// Mitsubishi GX Works2 project: GAO-71UR-20100027-0427R   PLC: Q00U

PROGRAM MAIN
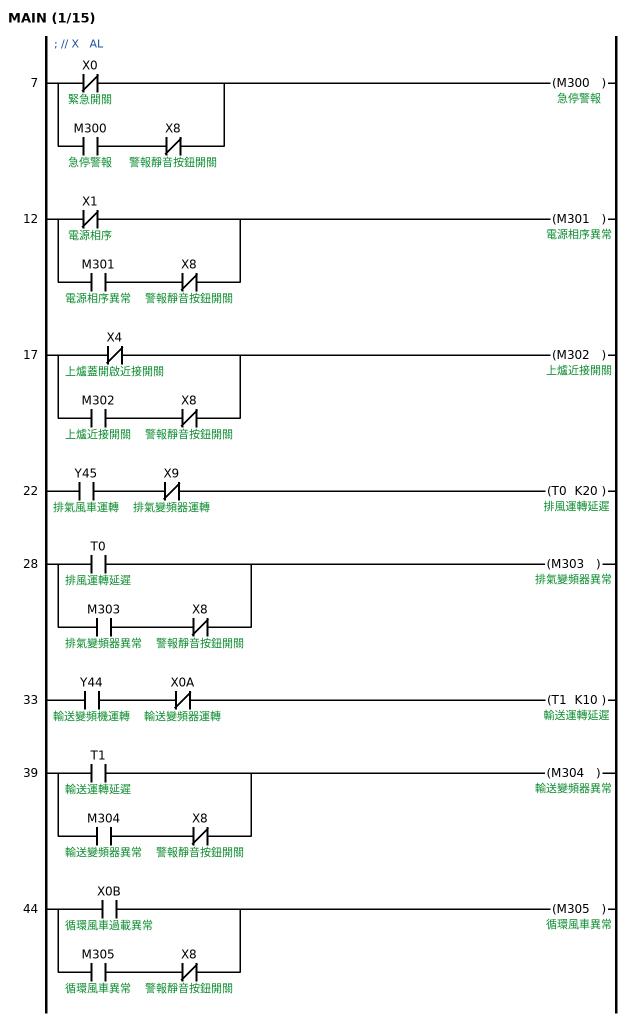
; // X   AL
7     LDI     X0  ; 緊急開關
      LD      M300  ; 急停警報
      ANI     X8  ; 警報靜音按鈕開關
      ORB
      OUT     M300  ; 急停警報
12    LDI     X1  ; 電源相序
      LD      M301  ; 電源相序異常
      ANI     X8  ; 警報靜音按鈕開關
      ORB
      OUT     M301  ; 電源相序異常
17    LDI     X4  ; 上爐蓋開啟近接開關
      LD      M302  ; 上爐近接開關
      ANI     X8  ; 警報靜音按鈕開關
      ORB
      OUT     M302  ; 上爐近接開關
22    LD      Y45  ; 排氣風車運轉
      ANI     X9  ; 排氣變頻器運轉
      OUT     T0 K20  ; 排風運轉延遲
28    LD      T0  ; 排風運轉延遲
      LD      M303  ; 排氣變頻器異常
      ANI     X8  ; 警報靜音按鈕開關
      ORB
      OUT     M303  ; 排氣變頻器異常
33    LD      Y44  ; 輸送變頻機運轉
      ANI     X0A  ; 輸送變頻器運轉
      OUT     T1 K10  ; 輸送運轉延遲
39    LD      T1  ; 輸送運轉延遲
      LD      M304  ; 輸送變頻器異常
      ANI     X8  ; 警報靜音按鈕開關
      ORB
      OUT     M304  ; 輸送變頻器異常
44    LD      X0B  ; 循環風車過載異常
      LD      M305  ; 循環風車異常
      ANI     X8  ; 警報靜音按鈕開關
      ORB
      OUT     M305  ; 循環風車異常
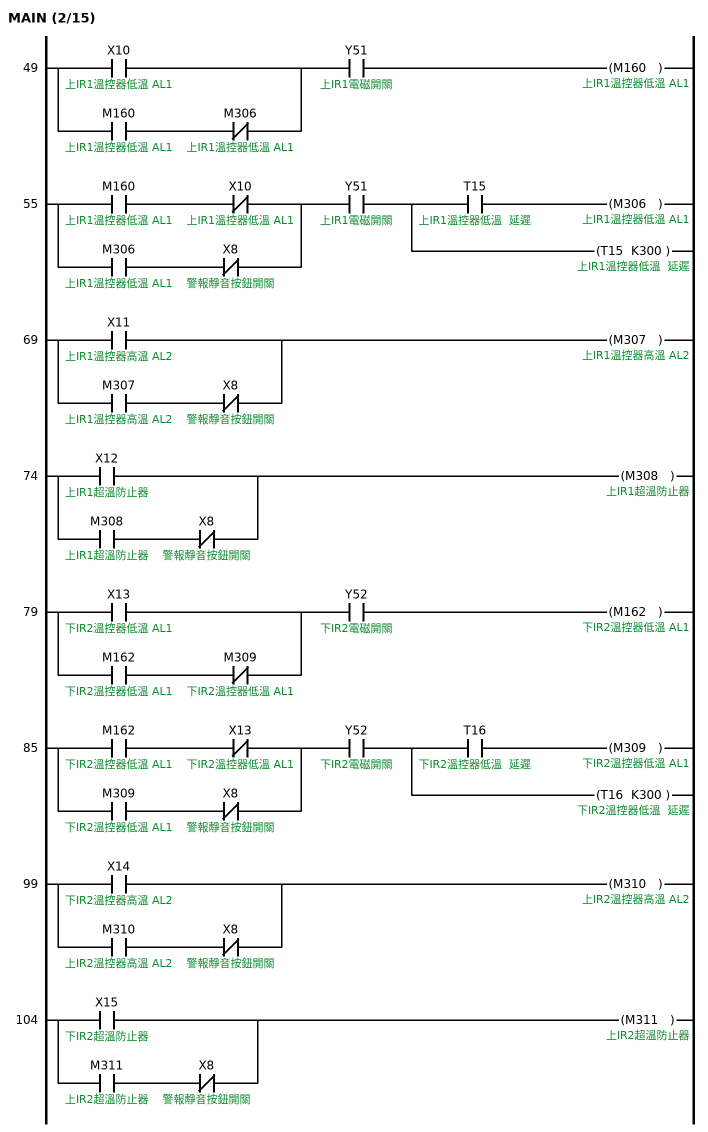
49    LD      X10  ; 上IR1溫控器低溫 AL1
      LD      M160  ; 上IR1溫控器低溫 AL1
      ANI     M306  ; 上IR1溫控器低溫 AL1
      ORB
      AND     Y51  ; 上IR1電磁開關
      OUT     M160  ; 上IR1溫控器低溫 AL1
55    LD      M160  ; 上IR1溫控器低溫 AL1
      ANI     X10  ; 上IR1溫控器低溫 AL1
      LD      M306  ; 上IR1溫控器低溫 AL1
      ANI     X8  ; 警報靜音按鈕開關
      ORB
      AND     Y51  ; 上IR1電磁開關
      MPS
      AND     T15  ; 上IR1溫控器低溫  延遲
      OUT     M306  ; 上IR1溫控器低溫 AL1
      MPP
      OUT     T15 K300  ; 上IR1溫控器低溫  延遲
69    LD      X11  ; 上IR1溫控器高溫 AL2
      LD      M307  ; 上IR1溫控器高溫 AL2
      ANI     X8  ; 警報靜音按鈕開關
      ORB
      OUT     M307  ; 上IR1溫控器高溫 AL2
74    LD      X12  ; 上IR1超溫防止器
      LD      M308  ; 上IR1超溫防止器
      ANI     X8  ; 警報靜音按鈕開關
      ORB
      OUT     M308  ; 上IR1超溫防止器
79    LD      X13  ; 下IR2溫控器低溫 AL1
      LD      M162  ; 下IR2溫控器低溫 AL1
      ANI     M309  ; 下IR2溫控器低溫 AL1
      ORB
      AND     Y52  ; 下IR2電磁開關
      OUT     M162  ; 下IR2溫控器低溫 AL1
85    LD      M162  ; 下IR2溫控器低溫 AL1
      ANI     X13  ; 下IR2溫控器低溫 AL1
      LD      M309  ; 下IR2溫控器低溫 AL1
      ANI     X8  ; 警報靜音按鈕開關
      ORB
      AND     Y52  ; 下IR2電磁開關
      MPS
      AND     T16  ; 下IR2溫控器低溫  延遲
      OUT     M309  ; 下IR2溫控器低溫 AL1
      MPP
      OUT     T16 K300  ; 下IR2溫控器低溫  延遲
99    LD      X14  ; 下IR2溫控器高溫 AL2
      LD      M310  ; 上IR2溫控器高溫 AL2
      ANI     X8  ; 警報靜音按鈕開關
      ORB
      OUT     M310  ; 上IR2溫控器高溫 AL2
104   LD      X15  ; 下IR2超溫防止器
      LD      M311  ; 上IR2超溫防止器
      ANI     X8  ; 警報靜音按鈕開關
      ORB
      OUT     M311  ; 上IR2超溫防止器
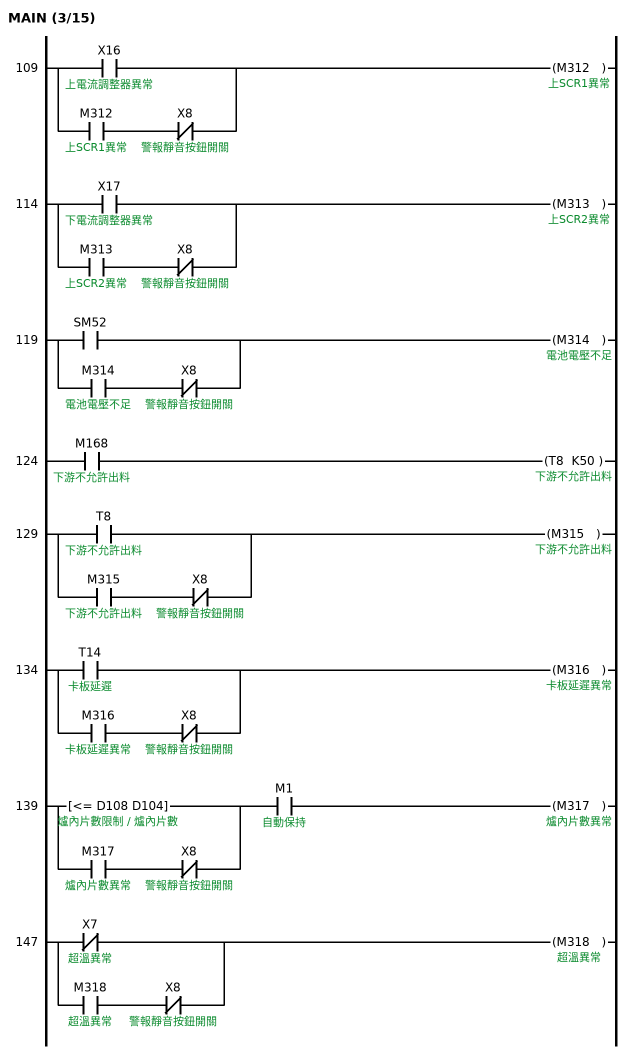
109   LD      X16  ; 上電流調整器異常
      LD      M312  ; 上SCR1異常
      ANI     X8  ; 警報靜音按鈕開關
      ORB
      OUT     M312  ; 上SCR1異常
114   LD      X17  ; 下電流調整器異常
      LD      M313  ; 上SCR2異常
      ANI     X8  ; 警報靜音按鈕開關
      ORB
      OUT     M313  ; 上SCR2異常
119   LD      SM52
      LD      M314  ; 電池電壓不足
      ANI     X8  ; 警報靜音按鈕開關
      ORB
      OUT     M314  ; 電池電壓不足
124   LD      M168  ; 下游不允許出料
      OUT     T8 K50  ; 下游不允許出料
129   LD      T8  ; 下游不允許出料
      LD      M315  ; 下游不允許出料
      ANI     X8  ; 警報靜音按鈕開關
      ORB
      OUT     M315  ; 下游不允許出料
134   LD      T14  ; 卡板延遲
      LD      M316  ; 卡板延遲異常
      ANI     X8  ; 警報靜音按鈕開關
      ORB
      OUT     M316  ; 卡板延遲異常
139   LD<=    D108 D104  ; 爐內片數限制 / 爐內片數
      LD      M317  ; 爐內片數異常
      ANI     X8  ; 警報靜音按鈕開關
      ORB
      AND     M1  ; 自動保持
      OUT     M317  ; 爐內片數異常
147   LDI     X7  ; 超溫異常
      LD      M318  ; 超溫異常
      ANI     X8  ; 警報靜音按鈕開關
      ORB
      OUT     M318  ; 超溫異常
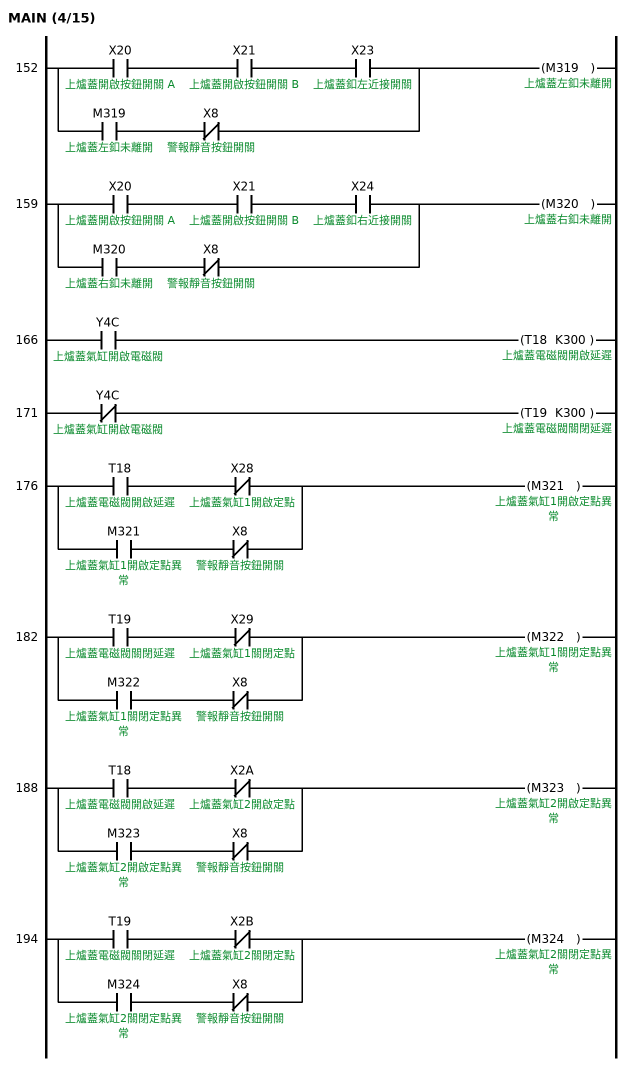
152   LD      X20  ; 上爐蓋開啟按鈕開關 A
      AND     X21  ; 上爐蓋開啟按鈕開關 B
      AND     X23  ; 上爐蓋釦左近接開關
      LD      M319  ; 上爐蓋左釦未離開
      ANI     X8  ; 警報靜音按鈕開關
      ORB
      OUT     M319  ; 上爐蓋左釦未離開
159   LD      X20  ; 上爐蓋開啟按鈕開關 A
      AND     X21  ; 上爐蓋開啟按鈕開關 B
      AND     X24  ; 上爐蓋釦右近接開關
      LD      M320  ; 上爐蓋右釦未離開
      ANI     X8  ; 警報靜音按鈕開關
      ORB
      OUT     M320  ; 上爐蓋右釦未離開
166   LD      Y4C  ; 上爐蓋氣缸開啟電磁閥
      OUT     T18 K300  ; 上爐蓋電磁閥開啟延遲
171   LDI     Y4C  ; 上爐蓋氣缸開啟電磁閥
      OUT     T19 K300  ; 上爐蓋電磁閥關閉延遲
176   LD      T18  ; 上爐蓋電磁閥開啟延遲
      ANI     X28  ; 上爐蓋氣缸1開啟定點
      LD      M321  ; 上爐蓋氣缸1開啟定點異常
      ANI     X8  ; 警報靜音按鈕開關
      ORB
      OUT     M321  ; 上爐蓋氣缸1開啟定點異常
182   LD      T19  ; 上爐蓋電磁閥關閉延遲
      ANI     X29  ; 上爐蓋氣缸1關閉定點
      LD      M322  ; 上爐蓋氣缸1關閉定點異常
      ANI     X8  ; 警報靜音按鈕開關
      ORB
      OUT     M322  ; 上爐蓋氣缸1關閉定點異常
188   LD      T18  ; 上爐蓋電磁閥開啟延遲
      ANI     X2A  ; 上爐蓋氣缸2開啟定點
      LD      M323  ; 上爐蓋氣缸2開啟定點異常
      ANI     X8  ; 警報靜音按鈕開關
      ORB
      OUT     M323  ; 上爐蓋氣缸2開啟定點異常
194   LD      T19  ; 上爐蓋電磁閥關閉延遲
      ANI     X2B  ; 上爐蓋氣缸2關閉定點
      LD      M324  ; 上爐蓋氣缸2關閉定點異常
      ANI     X8  ; 警報靜音按鈕開關
      ORB
      OUT     M324  ; 上爐蓋氣缸2關閉定點異常
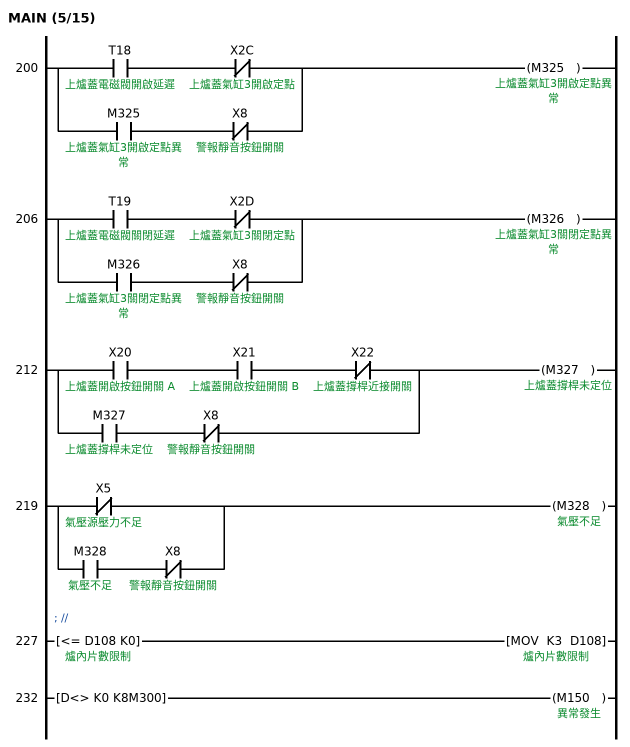
200   LD      T18  ; 上爐蓋電磁閥開啟延遲
      ANI     X2C  ; 上爐蓋氣缸3開啟定點
      LD      M325  ; 上爐蓋氣缸3開啟定點異常
      ANI     X8  ; 警報靜音按鈕開關
      ORB
      OUT     M325  ; 上爐蓋氣缸3開啟定點異常
206   LD      T19  ; 上爐蓋電磁閥關閉延遲
      ANI     X2D  ; 上爐蓋氣缸3關閉定點
      LD      M326  ; 上爐蓋氣缸3關閉定點異常
      ANI     X8  ; 警報靜音按鈕開關
      ORB
      OUT     M326  ; 上爐蓋氣缸3關閉定點異常
212   LD      X20  ; 上爐蓋開啟按鈕開關 A
      AND     X21  ; 上爐蓋開啟按鈕開關 B
      ANI     X22  ; 上爐蓋撐桿近接開關
      LD      M327  ; 上爐蓋撐桿未定位
      ANI     X8  ; 警報靜音按鈕開關
      ORB
      OUT     M327  ; 上爐蓋撐桿未定位
219   LDI     X5  ; 氣壓源壓力不足
      LD      M328  ; 氣壓不足
      ANI     X8  ; 警報靜音按鈕開關
      ORB
      OUT     M328  ; 氣壓不足
; //
227   LD<=    D108 K0  ; 爐內片數限制
      MOV     K3 D108
232   LDD<>   K0 K8M300  ; 急停警報
      OUT     M150  ; 異常發生
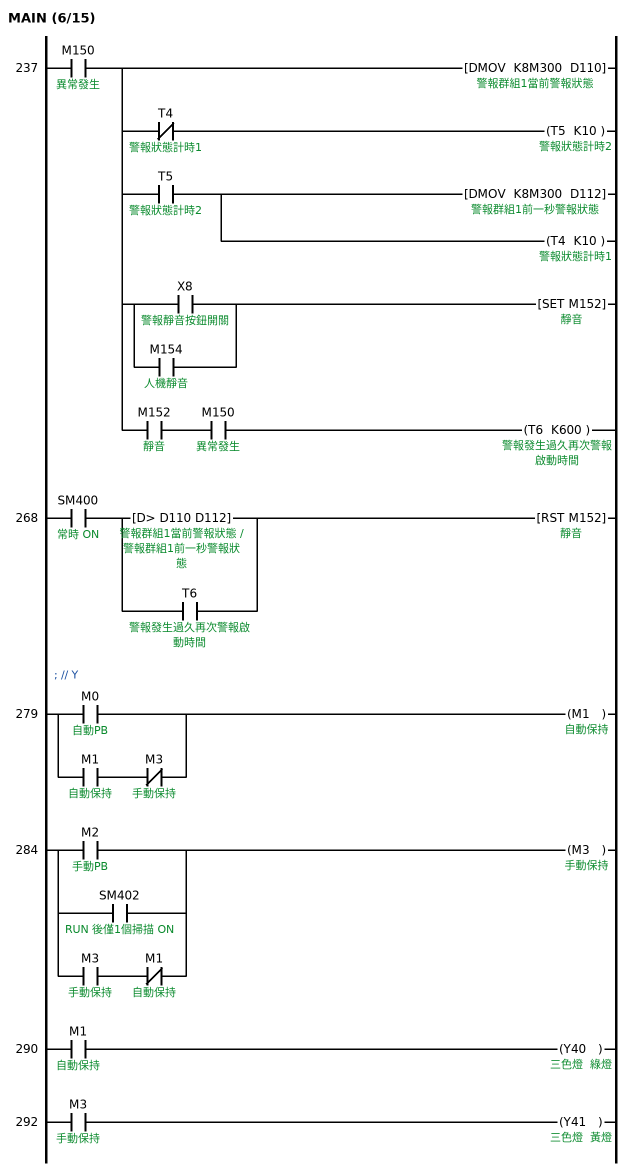
237   LD      M150  ; 異常發生
      DMOV    K8M300 D110  ; 警報群組1當前警報狀態
      MPS
      ANI     T4  ; 警報狀態計時1
      OUT     T5 K10  ; 警報狀態計時2
      MRD
      AND     T5  ; 警報狀態計時2
      DMOV    K8M300 D112  ; 警報群組1前一秒警報狀態
      OUT     T4 K10  ; 警報狀態計時1
      MRD
      LD      X8  ; 警報靜音按鈕開關
      OR      M154  ; 人機靜音
      ANB
      SET     M152  ; 靜音
      MPP
      AND     M152  ; 靜音
      AND     M150  ; 異常發生
      OUT     T6 K600  ; 警報發生過久再次警報啟動時間
268   LD      SM400  ; 常時 ON
      LDD>    D110 D112  ; 警報群組1當前警報狀態 / 警報群組1前一秒警報狀態
      OR      T6  ; 警報發生過久再次警報啟動時間
      ANB
      RST     M152  ; 靜音
; // Y
279   LD      M0  ; 自動PB
      LD      M1  ; 自動保持
      ANI     M3  ; 手動保持
      ORB
      OUT     M1  ; 自動保持
284   LD      M2  ; 手動PB
      OR      SM402  ; RUN 後僅1個掃描 ON
      LD      M3  ; 手動保持
      ANI     M1  ; 自動保持
      ORB
      OUT     M3  ; 手動保持
290   LD      M1  ; 自動保持
      OUT     Y40  ; 三色燈  綠燈
292   LD      M3  ; 手動保持
      OUT     Y41  ; 三色燈  黃燈
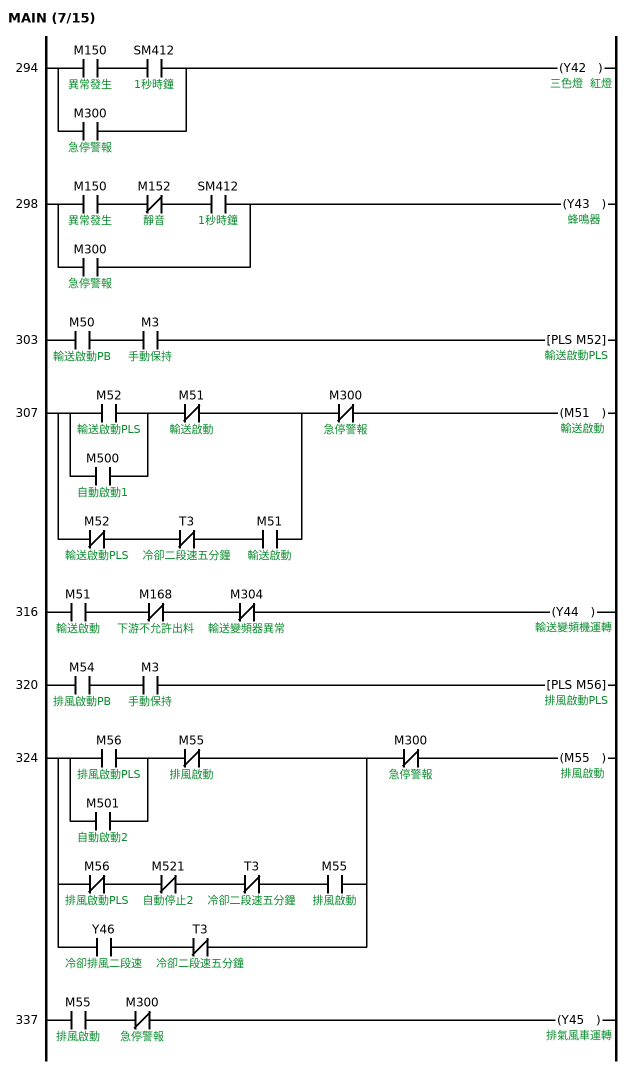
294   LD      M150  ; 異常發生
      AND     SM412  ; 1秒時鐘
      OR      M300  ; 急停警報
      OUT     Y42  ; 三色燈  紅燈
298   LD      M150  ; 異常發生
      ANI     M152  ; 靜音
      AND     SM412  ; 1秒時鐘
      OR      M300  ; 急停警報
      OUT     Y43  ; 蜂鳴器
303   LD      M50  ; 輸送啟動PB
      AND     M3  ; 手動保持
      PLS     M52  ; 輸送啟動PLS
307   LD      M52  ; 輸送啟動PLS
      OR      M500  ; 自動啟動1
      ANI     M51  ; 輸送啟動
      LDI     M52  ; 輸送啟動PLS
      ANI     T3  ; 冷卻二段速五分鐘
      AND     M51  ; 輸送啟動
      ORB
      ANI     M300  ; 急停警報
      OUT     M51  ; 輸送啟動
316   LD      M51  ; 輸送啟動
      ANI     M168  ; 下游不允許出料
      ANI     M304  ; 輸送變頻器異常
      OUT     Y44  ; 輸送變頻機運轉
320   LD      M54  ; 排風啟動PB
      AND     M3  ; 手動保持
      PLS     M56  ; 排風啟動PLS
324   LD      M56  ; 排風啟動PLS
      OR      M501  ; 自動啟動2
      ANI     M55  ; 排風啟動
      LDI     M56  ; 排風啟動PLS
      ANI     M521  ; 自動停止2
      ANI     T3  ; 冷卻二段速五分鐘
      AND     M55  ; 排風啟動
      ORB
      LD      Y46  ; 冷卻排風二段速
      ANI     T3  ; 冷卻二段速五分鐘
      ORB
      ANI     M300  ; 急停警報
      OUT     M55  ; 排風啟動
337   LD      M55  ; 排風啟動
      ANI     M300  ; 急停警報
      OUT     Y45  ; 排氣風車運轉
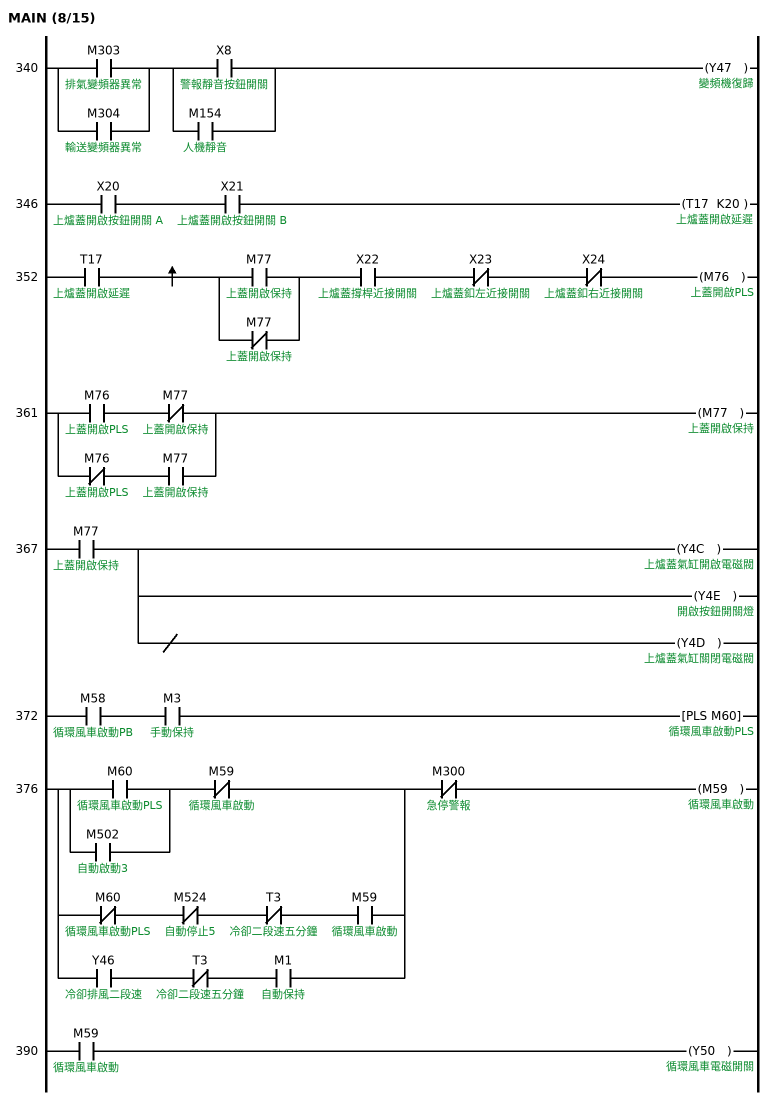
340   LD      M303  ; 排氣變頻器異常
      OR      M304  ; 輸送變頻器異常
      LD      X8  ; 警報靜音按鈕開關
      OR      M154  ; 人機靜音
      ANB
      OUT     Y47  ; 變頻機復歸
346   LD      X20  ; 上爐蓋開啟按鈕開關 A
      AND     X21  ; 上爐蓋開啟按鈕開關 B
      OUT     T17 K20  ; 上爐蓋開啟延遲
352   LD      T17  ; 上爐蓋開啟延遲
      MEP
      LD      M77  ; 上蓋開啟保持
      ORI     M77  ; 上蓋開啟保持
      ANB
      AND     X22  ; 上爐蓋撐桿近接開關
      ANI     X23  ; 上爐蓋釦左近接開關
      ANI     X24  ; 上爐蓋釦右近接開關
      OUT     M76  ; 上蓋開啟PLS
361   LD      M76  ; 上蓋開啟PLS
      ANI     M77  ; 上蓋開啟保持
      LDI     M76  ; 上蓋開啟PLS
      AND     M77  ; 上蓋開啟保持
      ORB
      OUT     M77  ; 上蓋開啟保持
367   LD      M77  ; 上蓋開啟保持
      OUT     Y4C  ; 上爐蓋氣缸開啟電磁閥
      OUT     Y4E  ; 開啟按鈕開關燈
      INV
      OUT     Y4D  ; 上爐蓋氣缸關閉電磁閥
372   LD      M58  ; 循環風車啟動PB
      AND     M3  ; 手動保持
      PLS     M60  ; 循環風車啟動PLS
376   LD      M60  ; 循環風車啟動PLS
      OR      M502  ; 自動啟動3
      ANI     M59  ; 循環風車啟動
      LDI     M60  ; 循環風車啟動PLS
      ANI     M524  ; 自動停止5
      ANI     T3  ; 冷卻二段速五分鐘
      AND     M59  ; 循環風車啟動
      ORB
      LD      Y46  ; 冷卻排風二段速
      ANI     T3  ; 冷卻二段速五分鐘
      AND     M1  ; 自動保持
      ORB
      ANI     M300  ; 急停警報
      OUT     M59  ; 循環風車啟動
390   LD      M59  ; 循環風車啟動
      OUT     Y50  ; 循環風車電磁開關
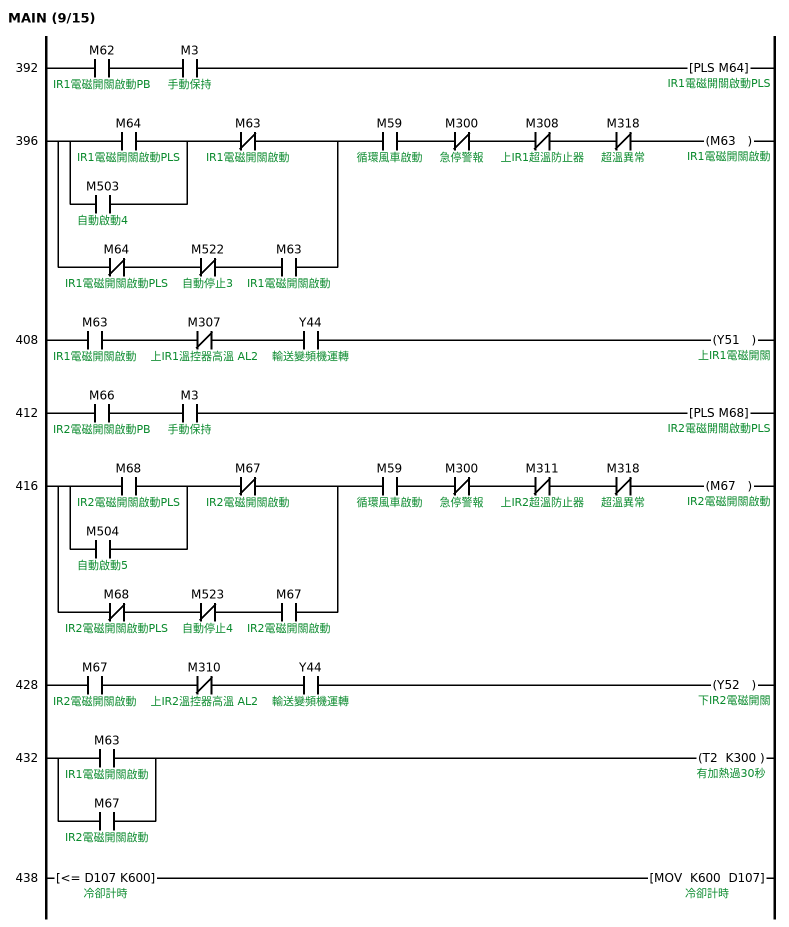
392   LD      M62  ; IR1電磁開關啟動PB
      AND     M3  ; 手動保持
      PLS     M64  ; IR1電磁開關啟動PLS
396   LD      M64  ; IR1電磁開關啟動PLS
      OR      M503  ; 自動啟動4
      ANI     M63  ; IR1電磁開關啟動
      LDI     M64  ; IR1電磁開關啟動PLS
      ANI     M522  ; 自動停止3
      AND     M63  ; IR1電磁開關啟動
      ORB
      AND     M59  ; 循環風車啟動
      ANI     M300  ; 急停警報
      ANI     M308  ; 上IR1超溫防止器
      ANI     M318  ; 超溫異常
      OUT     M63  ; IR1電磁開關啟動
408   LD      M63  ; IR1電磁開關啟動
      ANI     M307  ; 上IR1溫控器高溫 AL2
      AND     Y44  ; 輸送變頻機運轉
      OUT     Y51  ; 上IR1電磁開關
412   LD      M66  ; IR2電磁開關啟動PB
      AND     M3  ; 手動保持
      PLS     M68  ; IR2電磁開關啟動PLS
416   LD      M68  ; IR2電磁開關啟動PLS
      OR      M504  ; 自動啟動5
      ANI     M67  ; IR2電磁開關啟動
      LDI     M68  ; IR2電磁開關啟動PLS
      ANI     M523  ; 自動停止4
      AND     M67  ; IR2電磁開關啟動
      ORB
      AND     M59  ; 循環風車啟動
      ANI     M300  ; 急停警報
      ANI     M311  ; 上IR2超溫防止器
      ANI     M318  ; 超溫異常
      OUT     M67  ; IR2電磁開關啟動
428   LD      M67  ; IR2電磁開關啟動
      ANI     M310  ; 上IR2溫控器高溫 AL2
      AND     Y44  ; 輸送變頻機運轉
      OUT     Y52  ; 下IR2電磁開關
432   LD      M63  ; IR1電磁開關啟動
      OR      M67  ; IR2電磁開關啟動
      OUT     T2 K300  ; 有加熱過30秒
438   LD<=    D107 K600  ; 冷卻計時
      MOV     K600 D107
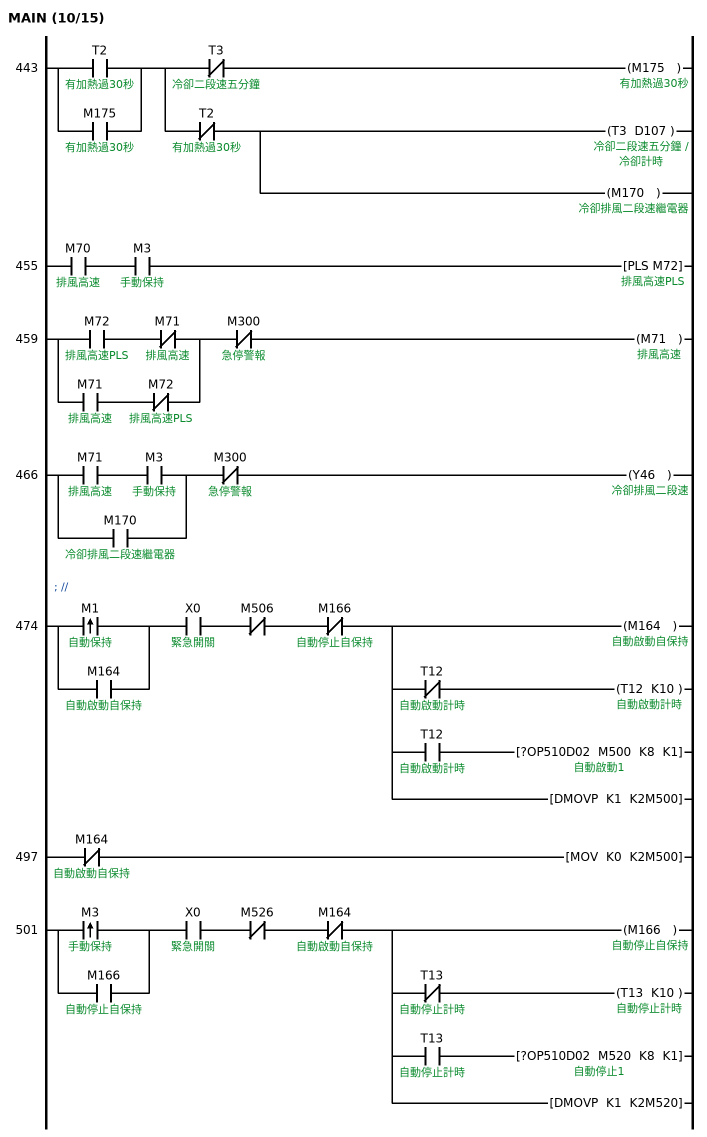
443   LD      T2  ; 有加熱過30秒
      OR      M175  ; 有加熱過30秒
      MPS
      ANI     T3  ; 冷卻二段速五分鐘
      OUT     M175  ; 有加熱過30秒
      MPP
      ANI     T2  ; 有加熱過30秒
      OUT     T3 D107  ; 冷卻二段速五分鐘 / 冷卻計時
      OUT     M170  ; 冷卻排風二段速繼電器
455   LD      M70  ; 排風高速
      AND     M3  ; 手動保持
      PLS     M72  ; 排風高速PLS
459   LD      M72  ; 排風高速PLS
      ANI     M71  ; 排風高速
      LD      M71  ; 排風高速
      ANI     M72  ; 排風高速PLS
      ORB
      ANI     M300  ; 急停警報
      OUT     M71  ; 排風高速
466   LD      M71  ; 排風高速
      AND     M3  ; 手動保持
      OR      M170  ; 冷卻排風二段速繼電器
      ANI     M300  ; 急停警報
      OUT     Y46  ; 冷卻排風二段速
; //
474   LDP     M1  ; 自動保持
      OR      M164  ; 自動啟動自保持
      AND     X0  ; 緊急開關
      ANI     M506
      ANI     M166  ; 自動停止自保持
      OUT     M164  ; 自動啟動自保持
      MPS
      ANI     T12  ; 自動啟動計時
      OUT     T12 K10  ; 自動啟動計時
      MRD
      AND     T12  ; 自動啟動計時
      ?OP510D02 M500 K8 K1
      MPP
      DMOVP   K1 K2M500
497   LDI     M164  ; 自動啟動自保持
      MOV     K0 K2M500
501   LDP     M3  ; 手動保持
      OR      M166  ; 自動停止自保持
      AND     X0  ; 緊急開關
      ANI     M526
      ANI     M164  ; 自動啟動自保持
      OUT     M166  ; 自動停止自保持
      MPS
      ANI     T13  ; 自動停止計時
      OUT     T13 K10  ; 自動停止計時
      MRD
      AND     T13  ; 自動停止計時
      ?OP510D02 M520 K8 K1  ; 自動停止1
      MPP
      DMOVP   K1 K2M520
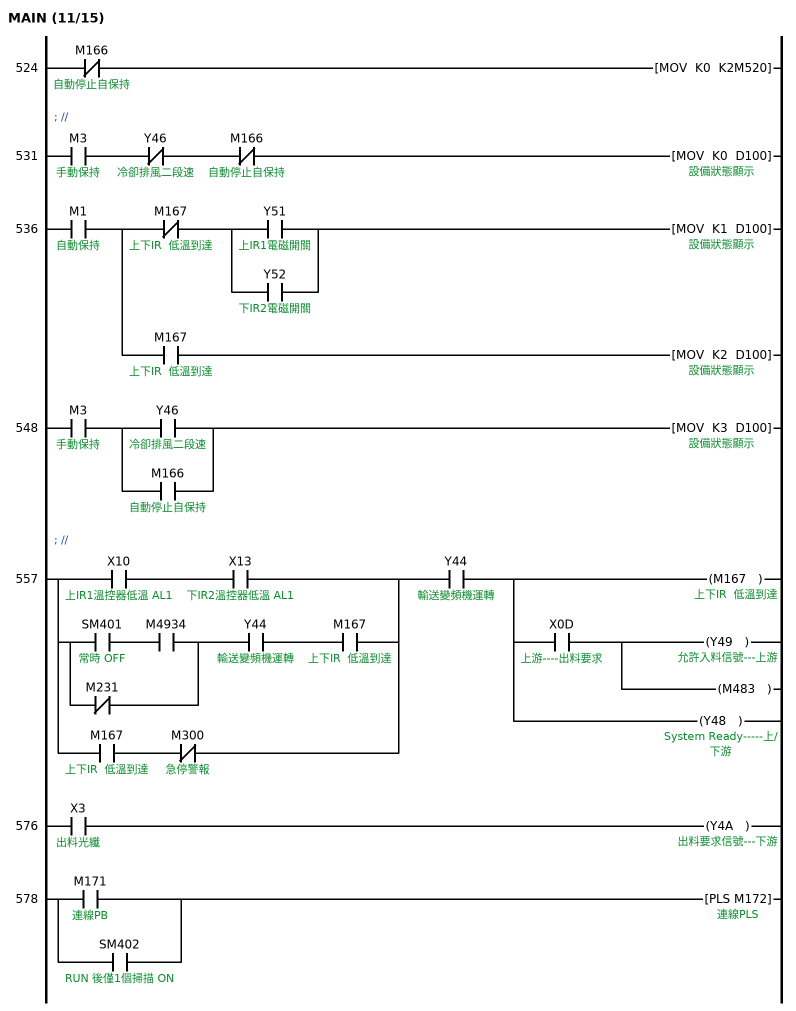
524   LDI     M166  ; 自動停止自保持
      MOV     K0 K2M520
; //
531   LD      M3  ; 手動保持
      ANI     Y46  ; 冷卻排風二段速
      ANI     M166  ; 自動停止自保持
      MOV     K0 D100  ; 設備狀態顯示
536   LD      M1  ; 自動保持
      MPS
      ANI     M167  ; 上下IR  低溫到達
      LD      Y51  ; 上IR1電磁開關
      OR      Y52  ; 下IR2電磁開關
      ANB
      MOV     K1 D100
      MPP
      AND     M167  ; 上下IR  低溫到達
      MOV     K2 D100
548   LD      M3  ; 手動保持
      LD      Y46  ; 冷卻排風二段速
      OR      M166  ; 自動停止自保持
      ANB
      MOV     K3 D100
; //
557   LD      X10  ; 上IR1溫控器低溫 AL1
      AND     X13  ; 下IR2溫控器低溫 AL1
      LD      SM401  ; 常時 OFF
      AND     M4934
      ORI     M231
      AND     Y44  ; 輸送變頻機運轉
      AND     M167  ; 上下IR  低溫到達
      ORB
      LD      M167  ; 上下IR  低溫到達
      ANI     M300  ; 急停警報
      ORB
      AND     Y44  ; 輸送變頻機運轉
      OUT     M167  ; 上下IR  低溫到達
      MPS
      AND     X0D  ; 上游----出料要求
      OUT     Y49  ; 允許入料信號---上游
      OUT     M483
      MPP
      OUT     Y48  ; System Ready-----上/下游
576   LD      X3  ; 出料光纖
      OUT     Y4A  ; 出料要求信號---下游
578   LD      M171  ; 連線PB
      OR      SM402  ; RUN 後僅1個掃描 ON
      PLS     M172  ; 連線PLS
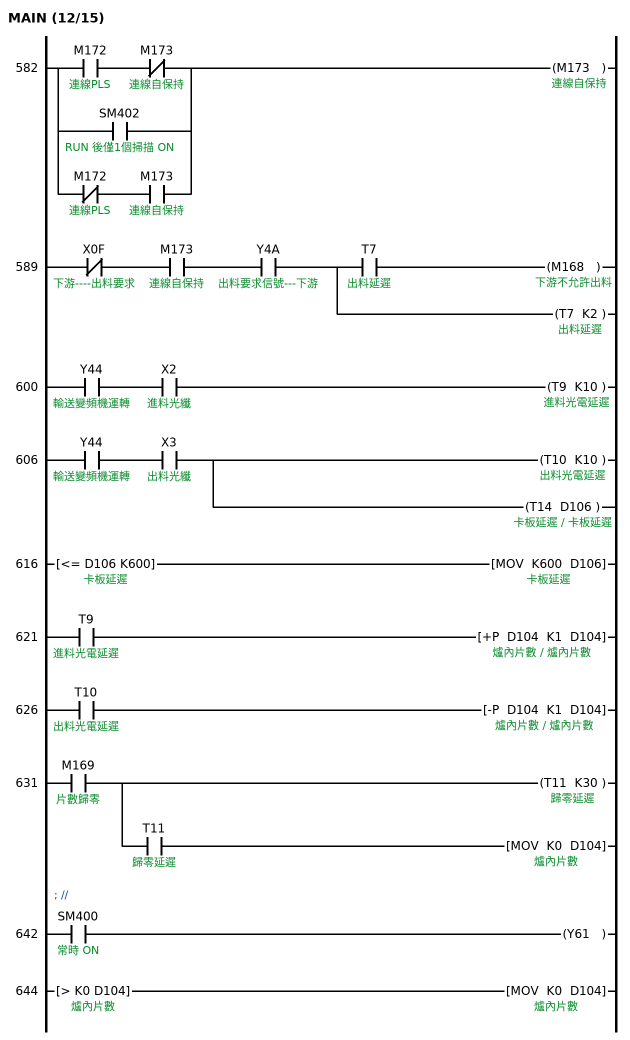
582   LD      M172  ; 連線PLS
      ANI     M173  ; 連線自保持
      OR      SM402  ; RUN 後僅1個掃描 ON
      LDI     M172  ; 連線PLS
      AND     M173  ; 連線自保持
      ORB
      OUT     M173  ; 連線自保持
589   LDI     X0F  ; 下游----出料要求
      AND     M173  ; 連線自保持
      AND     Y4A  ; 出料要求信號---下游
      MPS
      AND     T7  ; 出料延遲
      OUT     M168  ; 下游不允許出料
      MPP
      OUT     T7 K2  ; 出料延遲
600   LD      Y44  ; 輸送變頻機運轉
      AND     X2  ; 進料光纖
      OUT     T9 K10  ; 進料光電延遲
606   LD      Y44  ; 輸送變頻機運轉
      AND     X3  ; 出料光纖
      OUT     T10 K10  ; 出料光電延遲
      OUT     T14 D106  ; 卡板延遲 / 卡板延遲
616   LD<=    D106 K600  ; 卡板延遲
      MOV     K600 D106
621   LD      T9  ; 進料光電延遲
      +P      D104 K1 D104
626   LD      T10  ; 出料光電延遲
      -P      D104 K1 D104
631   LD      M169  ; 片數歸零
      OUT     T11 K30  ; 歸零延遲
      AND     T11  ; 歸零延遲
      MOV     K0 D104
; //
642   LD      SM400  ; 常時 ON
      OUT     Y61
644   LD>     K0 D104  ; 爐內片數
      MOV     K0 D104
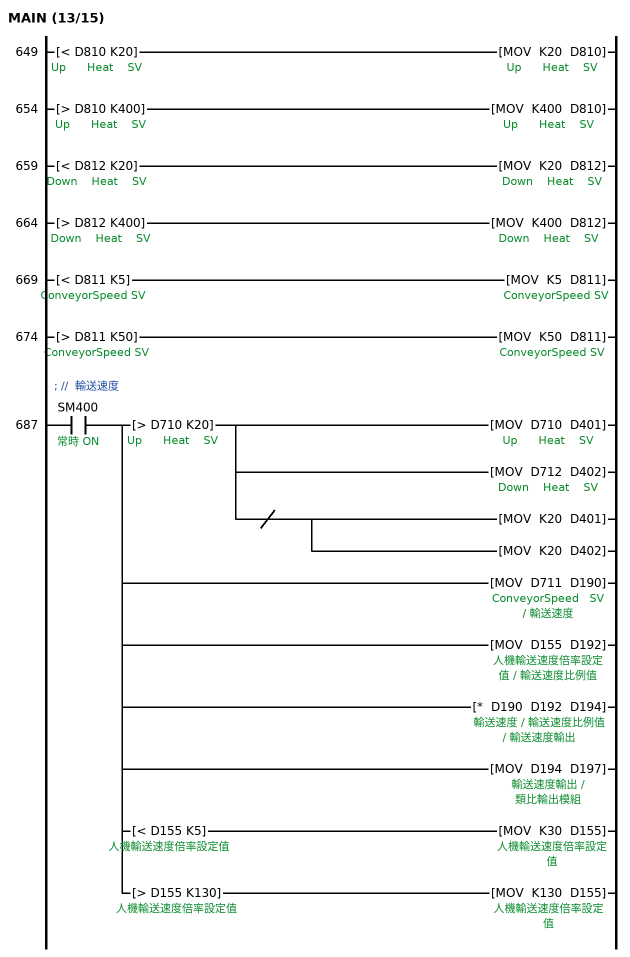
649   LD<     D810 K20  ; Up      Heat    SV
      MOV     K20 D810
654   LD>     D810 K400  ; Up      Heat    SV
      MOV     K400 D810
659   LD<     D812 K20  ; Down    Heat    SV
      MOV     K20 D812
664   LD>     D812 K400  ; Down    Heat    SV
      MOV     K400 D812
669   LD<     D811 K5  ; ConveyorSpeed SV
      MOV     K5 D811
674   LD>     D811 K50  ; ConveyorSpeed SV
      MOV     K50 D811
; //  輸送速度
687   LD      SM400  ; 常時 ON
      MPS
      AND>    D710 K20  ; Up      Heat    SV
      MOV     D710 D401
      MOV     D712 D402  ; Down    Heat    SV
      INV
      MOV     K20 D401
      MOV     K20 D402
      MPP
      MOV     D711 D190  ; ConveyorSpeed   SV / 輸送速度
      MOV     D155 D192  ; 人機輸送速度倍率設定值 / 輸送速度比例值
      *       D190 D192 D194  ; 輸送速度輸出
      MOV     D194 D197  ; 類比輸出模組
      MPS
      AND<    D155 K5  ; 人機輸送速度倍率設定值
      MOV     K30 D155
      MPP
      AND>    D155 K130  ; 人機輸送速度倍率設定值
      MOV     K130 D155
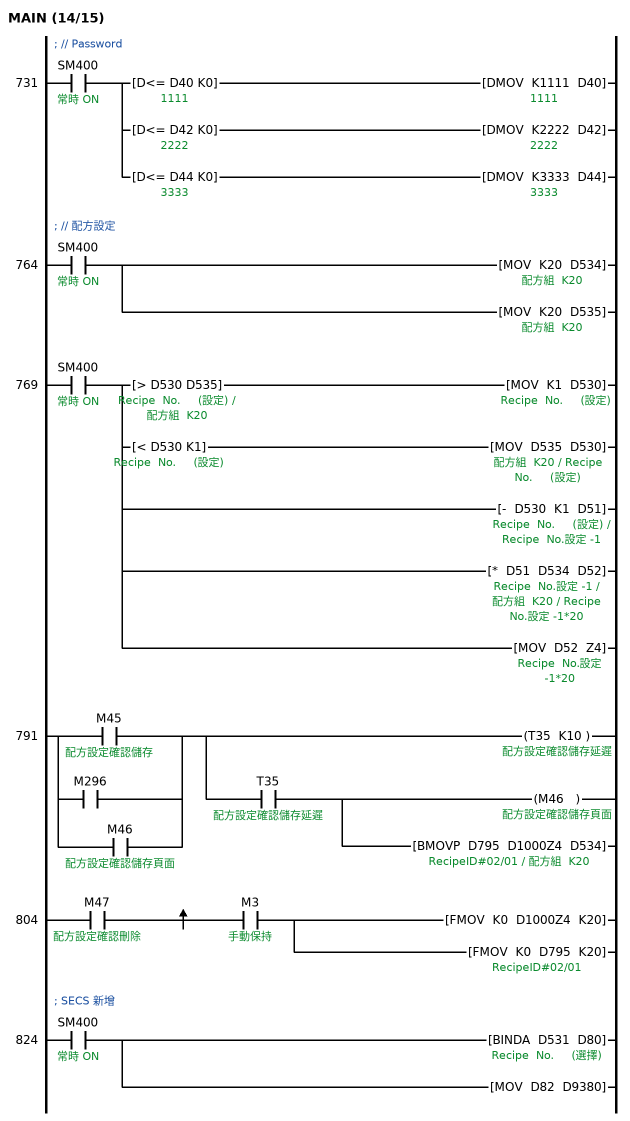
; // Password
731   LD      SM400  ; 常時 ON
      MPS
      ANDD<=  D40 K0  ; 1111
      DMOV    K1111 D40
      MRD
      ANDD<=  D42 K0  ; 2222
      DMOV    K2222 D42
      MPP
      ANDD<=  D44 K0  ; 3333
      DMOV    K3333 D44
; // 配方設定
764   LD      SM400  ; 常時 ON
      MOV     K20 D534  ; 配方組  K20
      MOV     K20 D535  ; 配方組  K20
769   LD      SM400  ; 常時 ON
      MPS
      AND>    D530 D535  ; Recipe  No.     (設定) / 配方組  K20
      MOV     K1 D530
      MRD
      AND<    D530 K1  ; Recipe  No.     (設定)
      MOV     D535 D530
      MPP
      -       D530 K1 D51  ; Recipe  No.設定 -1
      *       D51 D534 D52  ; Recipe  No.設定 -1*20
      MOV     D52 Z4
791   LD      M45  ; 配方設定確認儲存
      OR      M296
      OR      M46  ; 配方設定確認儲存頁面
      OUT     T35 K10  ; 配方設定確認儲存延遲
      AND     T35  ; 配方設定確認儲存延遲
      OUT     M46  ; 配方設定確認儲存頁面
      BMOVP   D795 D1000Z4 D534  ; RecipeID#02/01
804   LD      M47  ; 配方設定確認刪除
      MEP
      AND     M3  ; 手動保持
      FMOV    K0 D1000Z4 K20
      FMOV    K0 D795 K20
; SECS 新增
824   LD      SM400  ; 常時 ON
      BINDA   D531 D80  ; Recipe  No.     (選擇)
      MOV     D82 D9380
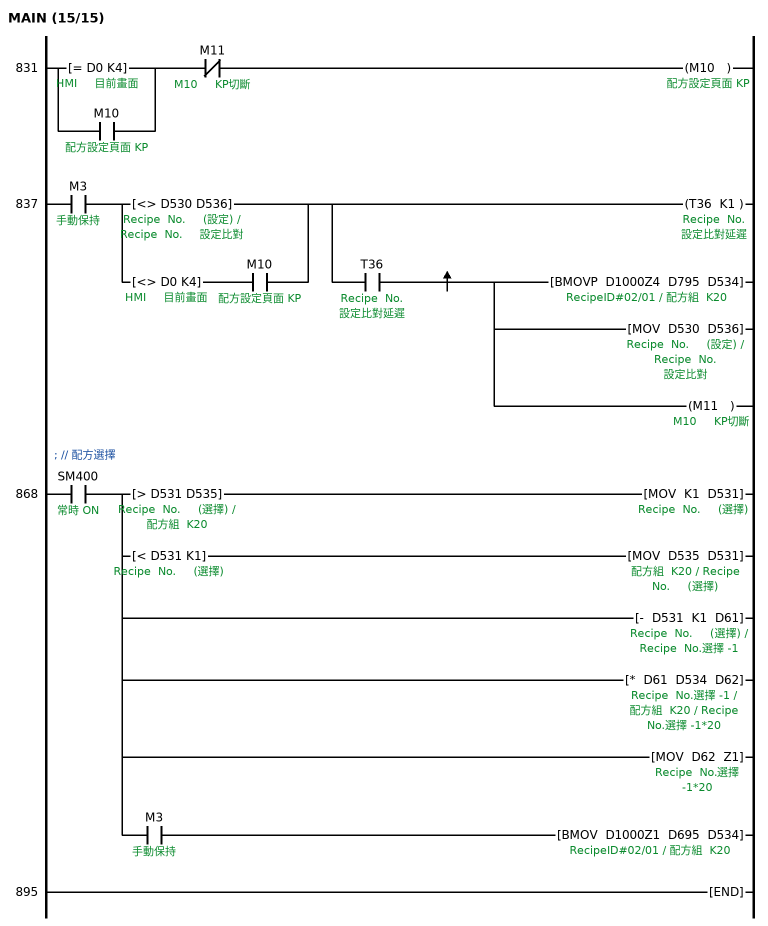
831   LD=     D0 K4  ; HMI     目前畫面
      OR      M10  ; 配方設定頁面 KP
      ANI     M11  ; M10     KP切斷
      OUT     M10  ; 配方設定頁面 KP
837   LD      M3  ; 手動保持
      LD<>    D530 D536  ; Recipe  No.     (設定) / Recipe  No.     設定比對
      LD<>    D0 K4  ; HMI     目前畫面
      AND     M10  ; 配方設定頁面 KP
      ORB
      ANB
      OUT     T36 K1  ; Recipe  No.     設定比對延遲
      AND     T36  ; Recipe  No.     設定比對延遲
      MEP
      BMOVP   D1000Z4 D795 D534
      MOV     D530 D536
      OUT     M11  ; M10     KP切斷
; // 配方選擇
868   LD      SM400  ; 常時 ON
      MPS
      AND>    D531 D535  ; Recipe  No.     (選擇) / 配方組  K20
      MOV     K1 D531
      MRD
      AND<    D531 K1  ; Recipe  No.     (選擇)
      MOV     D535 D531
      MPP
      -       D531 K1 D61  ; Recipe  No.選擇 -1
      *       D61 D534 D62  ; Recipe  No.選擇 -1*20
      MOV     D62 Z1
      AND     M3  ; 手動保持
      BMOV    D1000Z1 D695 D534  ; RecipeID#02/01
895   END
END_PROGRAM

PROGRAM SECS
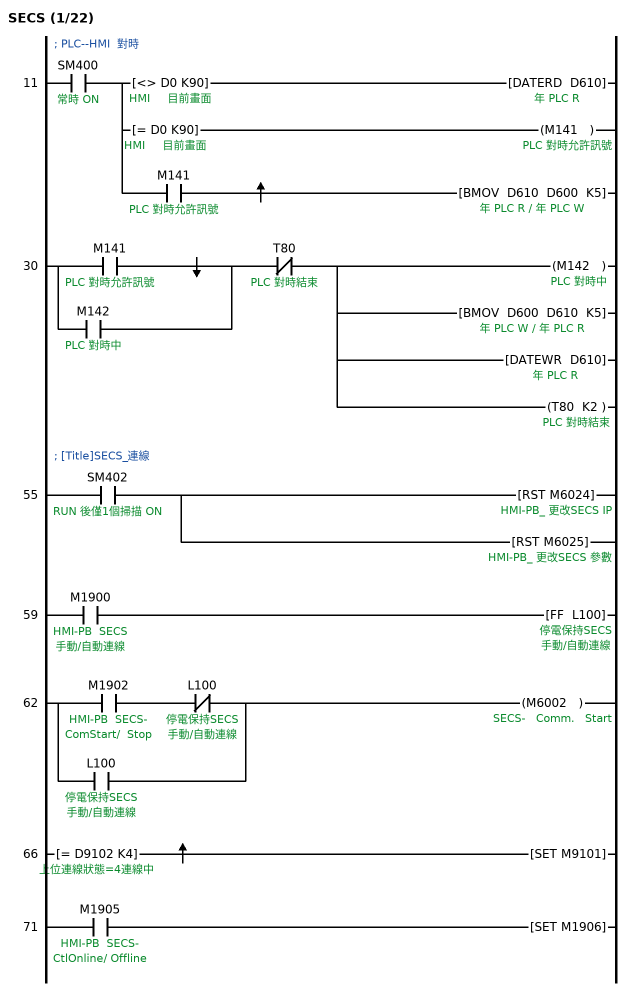
; PLC--HMI  對時
11    LD      SM400  ; 常時 ON
      MPS
      AND<>   D0 K90  ; HMI     目前畫面
      DATERD  D610  ; 年 PLC R
      MRD
      AND=    D0 K90  ; HMI     目前畫面
      OUT     M141  ; PLC 對時允許訊號
      MPP
      AND     M141  ; PLC 對時允許訊號
      MEP
      BMOV    D610 D600 K5  ; 年 PLC W
30    LD      M141  ; PLC 對時允許訊號
      MEF
      OR      M142  ; PLC 對時中
      ANI     T80  ; PLC 對時結束
      OUT     M142  ; PLC 對時中
      BMOV    D600 D610 K5
      DATEWR  D610
      OUT     T80 K2  ; PLC 對時結束
; [Title]SECS_連線
55    LD      SM402  ; RUN 後僅1個掃描 ON
      RST     M6024  ; HMI-PB_ 更改SECS IP
      RST     M6025  ; HMI-PB_ 更改SECS 參數
59    LD      M1900  ; HMI-PB  SECS    手動/自動連線
      FF      L100  ; 停電保持SECS    手動/自動連線
62    LD      M1902  ; HMI-PB  SECS-ComStart/  Stop
      ANI     L100  ; 停電保持SECS    手動/自動連線
      OR      L100  ; 停電保持SECS    手動/自動連線
      OUT     M6002  ; SECS-   Comm.   Start
66    LD=     D9102 K4  ; 上位連線狀態=4連線中
      MEP
      SET     M9101
71    LD      M1905  ; HMI-PB  SECS-CtlOnline/ Offline
      SET     M1906
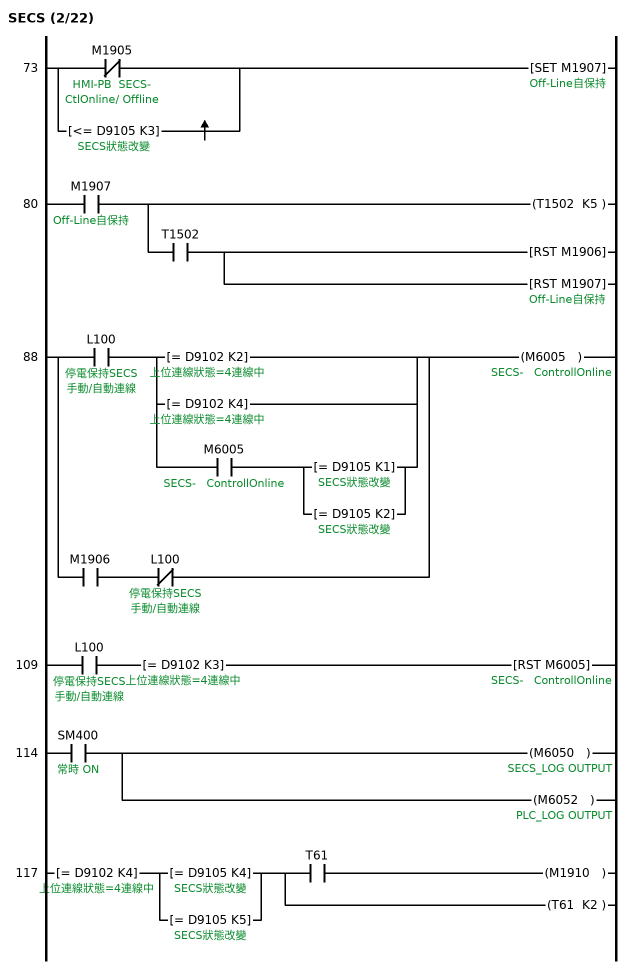
73    LDI     M1905  ; HMI-PB  SECS-CtlOnline/ Offline
      LD<=    D9105 K3  ; SECS狀態改變
      MEP
      ORB
      SET     M1907  ; Off-Line自保持
80    LD      M1907  ; Off-Line自保持
      OUT     T1502 K5
      AND     T1502
      RST     M1906
      RST     M1907  ; Off-Line自保持
88    LD      L100  ; 停電保持SECS    手動/自動連線
      LD=     D9102 K2  ; 上位連線狀態=4連線中
      OR=     D9102 K4  ; 上位連線狀態=4連線中
      LD      M6005  ; SECS-   ControllOnline
      LD=     D9105 K1  ; SECS狀態改變
      OR=     D9105 K2  ; SECS狀態改變
      ANB
      ORB
      ANB
      LD      M1906
      ANI     L100  ; 停電保持SECS    手動/自動連線
      ORB
      OUT     M6005  ; SECS-   ControllOnline
109   LD      L100  ; 停電保持SECS    手動/自動連線
      AND=    D9102 K3  ; 上位連線狀態=4連線中
      RST     M6005  ; SECS-   ControllOnline
114   LD      SM400  ; 常時 ON
      OUT     M6050  ; SECS_LOG OUTPUT
      OUT     M6052  ; PLC_LOG OUTPUT
117   LD=     D9102 K4  ; 上位連線狀態=4連線中
      LD=     D9105 K4  ; SECS狀態改變
      OR=     D9105 K5  ; SECS狀態改變
      ANB
      MPS
      AND     T61
      OUT     M1910
      MPP
      OUT     T61 K2
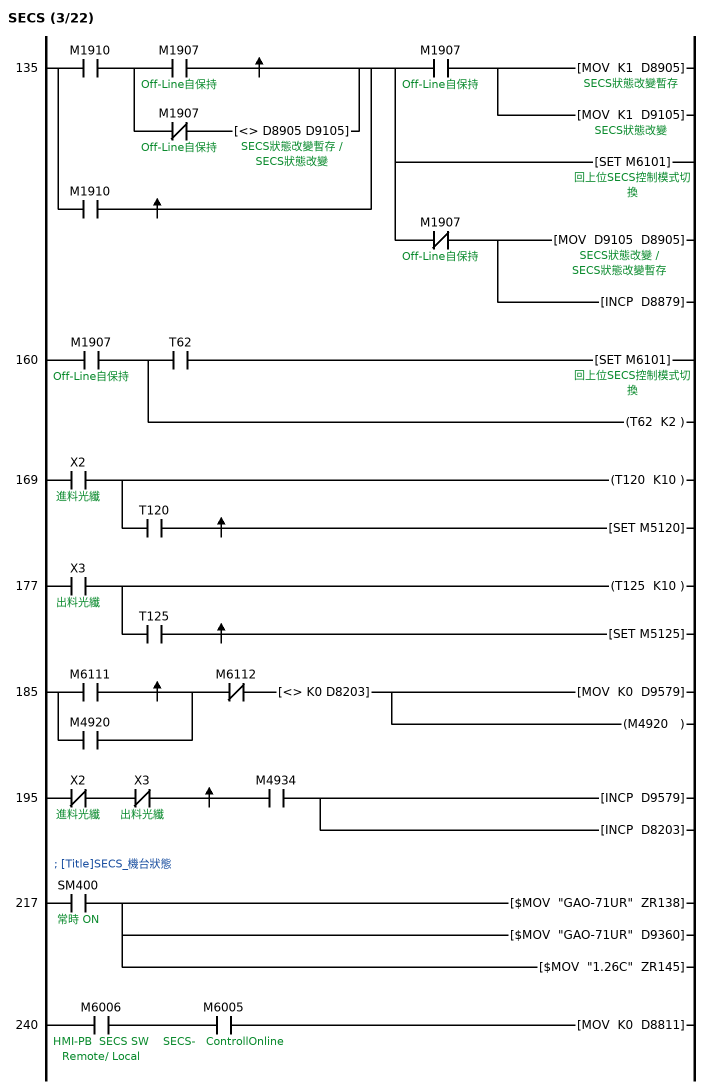
135   LD      M1910
      LD      M1907  ; Off-Line自保持
      MEP
      LDI     M1907  ; Off-Line自保持
      AND<>   D8905 D9105  ; SECS狀態改變暫存 / SECS狀態改變
      ORB
      ANB
      LD      M1910
      MEP
      ORB
      MPS
      AND     M1907  ; Off-Line自保持
      MOV     K1 D8905
      MOV     K1 D9105
      MPP
      SET     M6101  ; 回上位SECS控制模式切換
      ANI     M1907  ; Off-Line自保持
      MOV     D9105 D8905
      INCP    D8879
160   LD      M1907  ; Off-Line自保持
      MPS
      AND     T62
      SET     M6101  ; 回上位SECS控制模式切換
      MPP
      OUT     T62 K2
169   LD      X2  ; 進料光纖
      OUT     T120 K10
      AND     T120
      MEP
      SET     M5120
177   LD      X3  ; 出料光纖
      OUT     T125 K10
      AND     T125
      MEP
      SET     M5125
185   LD      M6111
      MEP
      OR      M4920
      ANI     M6112
      AND<>   K0 D8203
      MOV     K0 D9579
      OUT     M4920
195   LDI     X2  ; 進料光纖
      ANI     X3  ; 出料光纖
      MEP
      AND     M4934
      INCP    D9579
      INCP    D8203
; [Title]SECS_機台狀態
217   LD      SM400  ; 常時 ON
      $MOV    "GAO-71UR" ZR138
      $MOV    "GAO-71UR" D9360
      $MOV    "1.26C" ZR145
240   LD      M6006  ; HMI-PB  SECS SW  Remote/ Local
      AND     M6005  ; SECS-   ControllOnline
      MOV     K0 D8811
        [note] D8811=K0(遠程控制+SEC在線中)
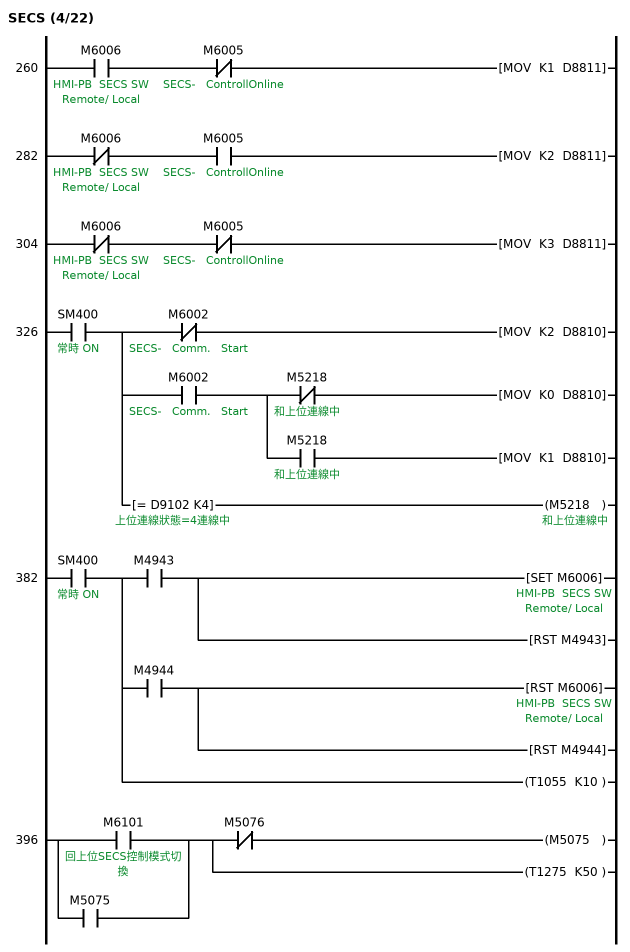
260   LD      M6006  ; HMI-PB  SECS SW  Remote/ Local
      ANI     M6005  ; SECS-   ControllOnline
      MOV     K1 D8811
        [note] D8811= k1(遠程控制中+SEC離線中)
282   LDI     M6006  ; HMI-PB  SECS SW  Remote/ Local
      AND     M6005  ; SECS-   ControllOnline
      MOV     K2 D8811
        [note] D881=k2(遠程控制離線+SEC在線中)
304   LDI     M6006  ; HMI-PB  SECS SW  Remote/ Local
      ANI     M6005  ; SECS-   ControllOnline
      MOV     K3 D8811
        [note] D881=k3(遠程控制離線+SEC離線中)
326   LD      SM400  ; 常時 ON
      MPS
      ANI     M6002  ; SECS-   Comm.   Start
      MOV     K2 D8810
        [note] K2= SEC通訊未連線
      MRD
      AND     M6002  ; SECS-   Comm.   Start
      MPS
      ANI     M5218  ; 和上位連線中
      MOV     K0 D8810
        [note] K0=SEC連線---上位未連線
      MPP
      AND     M5218  ; 和上位連線中
      MOV     K1 D8810
        [note] K1=SEC和上位連線中
      MPP
      AND=    D9102 K4  ; 上位連線狀態=4連線中
      OUT     M5218  ; 和上位連線中
382   LD      SM400  ; 常時 ON
      MPS
      AND     M4943
      SET     M6006  ; HMI-PB  SECS SW  Remote/ Local
      RST     M4943
      MRD
      AND     M4944
      RST     M6006  ; HMI-PB  SECS SW  Remote/ Local
      RST     M4944
      MPP
      OUT     T1055 K10
396   LD      M6101  ; 回上位SECS控制模式切換
      OR      M5075
      MPS
      ANI     M5076
      OUT     M5075
      MPP
      OUT     T1275 K50
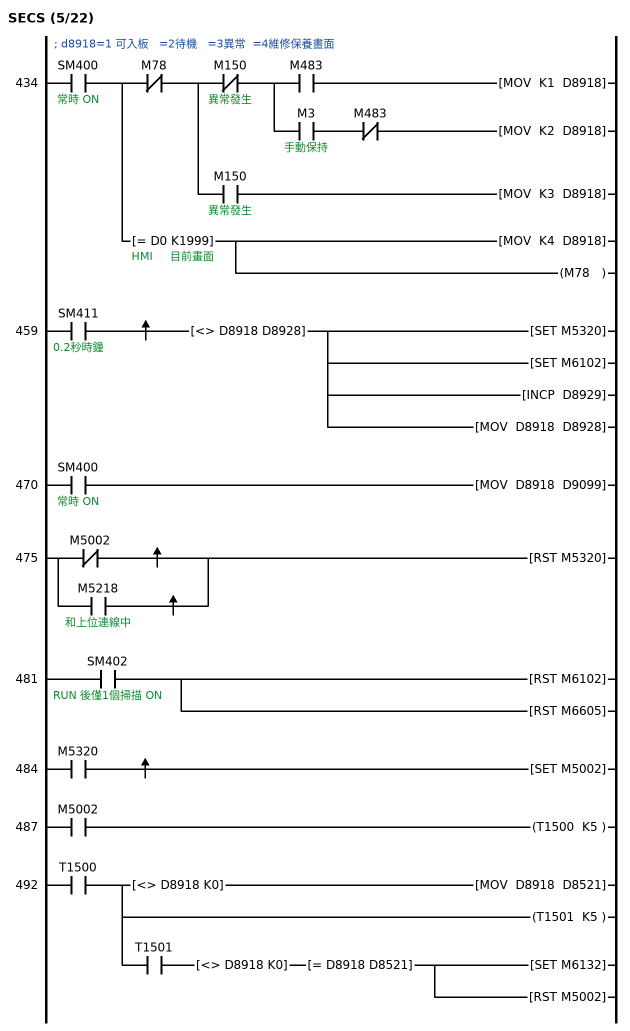
; d8918=1 可入板   =2待機   =3異常  =4維修保養畫面
434   LD      SM400  ; 常時 ON
      MPS
      ANI     M78
      MPS
      ANI     M150  ; 異常發生
      MPS
      AND     M483
      MOV     K1 D8918
      MPP
      AND     M3  ; 手動保持
      ANI     M483
      MOV     K2 D8918
      MPP
      AND     M150  ; 異常發生
      MOV     K3 D8918
      MPP
      AND=    D0 K1999  ; HMI     目前畫面
      MOV     K4 D8918
      OUT     M78
459   LD      SM411  ; 0.2秒時鐘
      MEP
      AND<>   D8918 D8928
      SET     M5320
      SET     M6102
      INCP    D8929
      MOV     D8918 D8928
470   LD      SM400  ; 常時 ON
      MOV     D8918 D9099
475   LDI     M5002
      MEP
      LD      M5218  ; 和上位連線中
      MEP
      ORB
      RST     M5320
481   LD      SM402  ; RUN 後僅1個掃描 ON
      RST     M6102
      RST     M6605
484   LD      M5320
      MEP
      SET     M5002
487   LD      M5002
      OUT     T1500 K5
492   LD      T1500
      MPS
      AND<>   D8918 K0
      MOV     D8918 D8521
      MPP
      OUT     T1501 K5
      AND     T1501
      AND<>   D8918 K0
      AND=    D8918 D8521
      SET     M6132
      RST     M5002
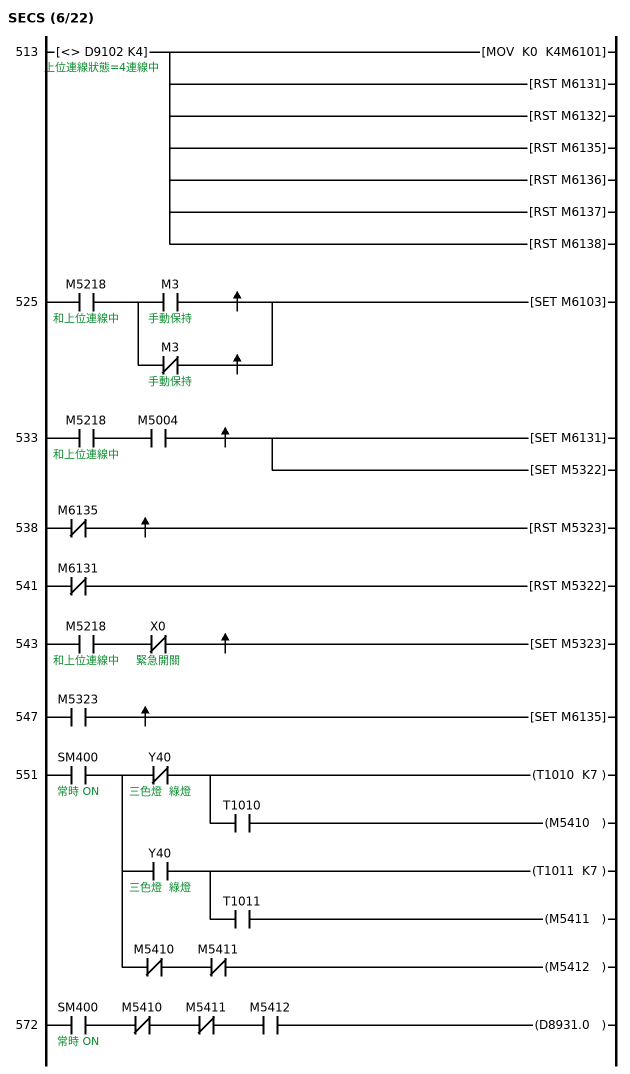
513   LD<>    D9102 K4  ; 上位連線狀態=4連線中
      MOV     K0 K4M6101
      RST     M6131
      RST     M6132
      RST     M6135
      RST     M6136
      RST     M6137
      RST     M6138
525   LD      M5218  ; 和上位連線中
      LD      M3  ; 手動保持
      MEP
      LDI     M3  ; 手動保持
      MEP
      ORB
      ANB
      SET     M6103
533   LD      M5218  ; 和上位連線中
      AND     M5004
      MEP
      SET     M6131
      SET     M5322
538   LDI     M6135
      MEP
      RST     M5323
541   LDI     M6131
      RST     M5322
543   LD      M5218  ; 和上位連線中
      ANI     X0  ; 緊急開關
      MEP
      SET     M5323
547   LD      M5323
      MEP
      SET     M6135
551   LD      SM400  ; 常時 ON
      MPS
      ANI     Y40  ; 三色燈  綠燈
      OUT     T1010 K7
      AND     T1010
      OUT     M5410
      MRD
      AND     Y40  ; 三色燈  綠燈
      OUT     T1011 K7
      AND     T1011
      OUT     M5411
      MPP
      ANI     M5410
      ANI     M5411
      OUT     M5412
572   LD      SM400  ; 常時 ON
      ANI     M5410
      ANI     M5411
      AND     M5412
      OUT     D8931.0
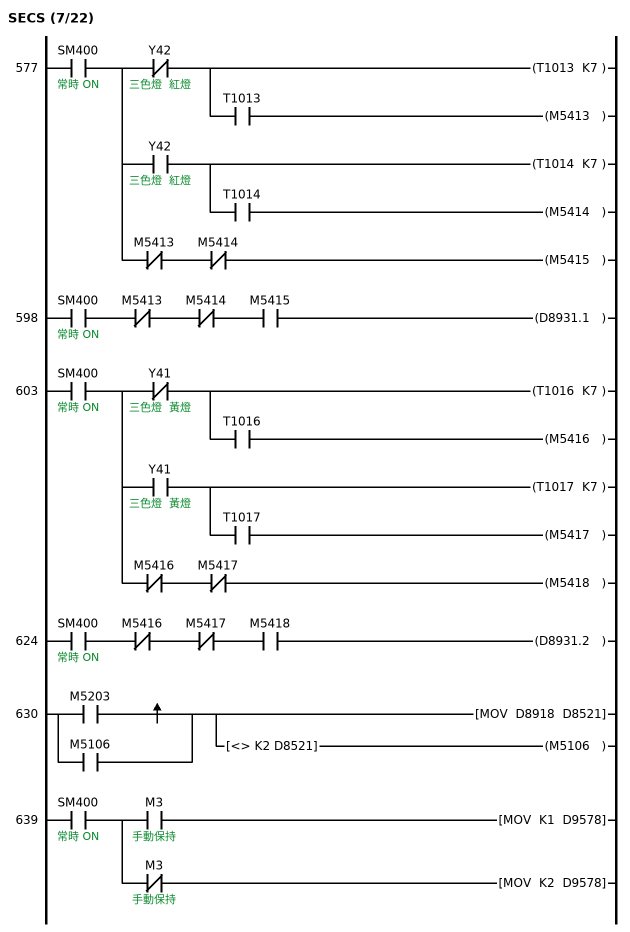
577   LD      SM400  ; 常時 ON
      MPS
      ANI     Y42  ; 三色燈  紅燈
      OUT     T1013 K7
      AND     T1013
      OUT     M5413
      MRD
      AND     Y42  ; 三色燈  紅燈
      OUT     T1014 K7
      AND     T1014
      OUT     M5414
      MPP
      ANI     M5413
      ANI     M5414
      OUT     M5415
598   LD      SM400  ; 常時 ON
      ANI     M5413
      ANI     M5414
      AND     M5415
      OUT     D8931.1
603   LD      SM400  ; 常時 ON
      MPS
      ANI     Y41  ; 三色燈  黃燈
      OUT     T1016 K7
      AND     T1016
      OUT     M5416
      MRD
      AND     Y41  ; 三色燈  黃燈
      OUT     T1017 K7
      AND     T1017
      OUT     M5417
      MPP
      ANI     M5416
      ANI     M5417
      OUT     M5418
624   LD      SM400  ; 常時 ON
      ANI     M5416
      ANI     M5417
      AND     M5418
      OUT     D8931.2
630   LD      M5203
      MEP
      OR      M5106
      MOV     D8918 D8521
      AND<>   K2 D8521
      OUT     M5106
639   LD      SM400  ; 常時 ON
      MPS
      AND     M3  ; 手動保持
      MOV     K1 D9578
      MPP
      ANI     M3  ; 手動保持
      MOV     K2 D9578
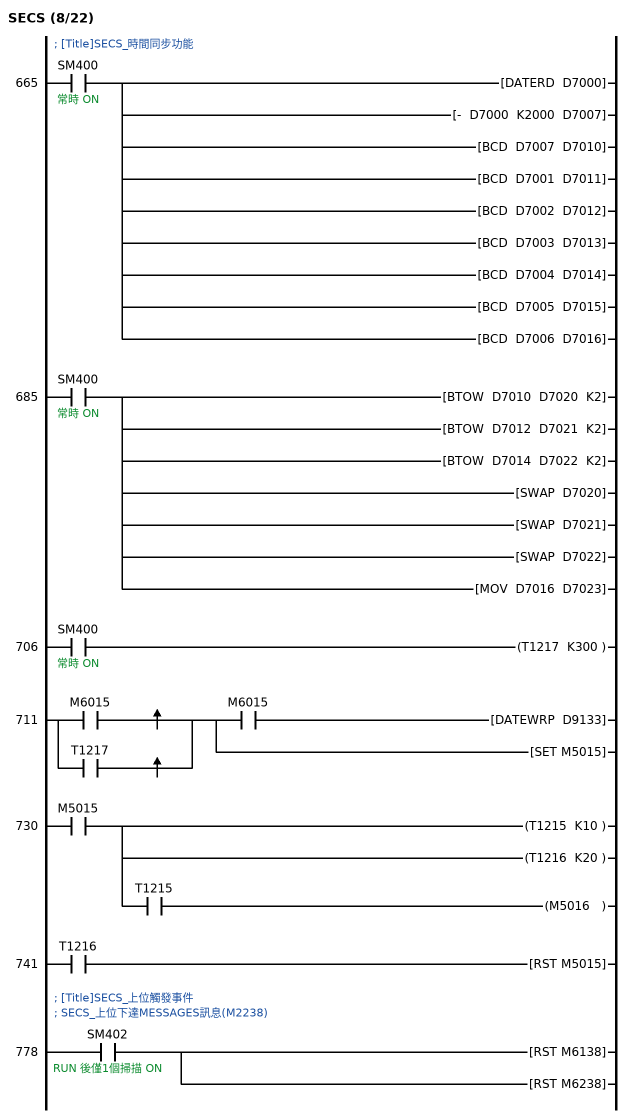
; [Title]SECS_時間同步功能
665   LD      SM400  ; 常時 ON
      DATERD  D7000
      -       D7000 K2000 D7007
      BCD     D7007 D7010
      BCD     D7001 D7011
      BCD     D7002 D7012
      BCD     D7003 D7013
      BCD     D7004 D7014
      BCD     D7005 D7015
      BCD     D7006 D7016
685   LD      SM400  ; 常時 ON
      BTOW    D7010 D7020 K2
      BTOW    D7012 D7021 K2
      BTOW    D7014 D7022 K2
      SWAP    D7020
      SWAP    D7021
      SWAP    D7022
      MOV     D7016 D7023
706   LD      SM400  ; 常時 ON
      OUT     T1217 K300
711   LD      M6015
      MEP
      LD      T1217
      MEP
      ORB
      MPS
      AND     M6015
      DATEWRP D9133
        [note] 寫入時間指令
      MPP
      SET     M5015
730   LD      M5015
      OUT     T1215 K10
      OUT     T1216 K20
      AND     T1215
      OUT     M5016
741   LD      T1216
      RST     M5015
; [Title]SECS_上位觸發事件
; SECS_上位下達MESSAGES訊息(M2238)
778   LD      SM402  ; RUN 後僅1個掃描 ON
      RST     M6138
      RST     M6238
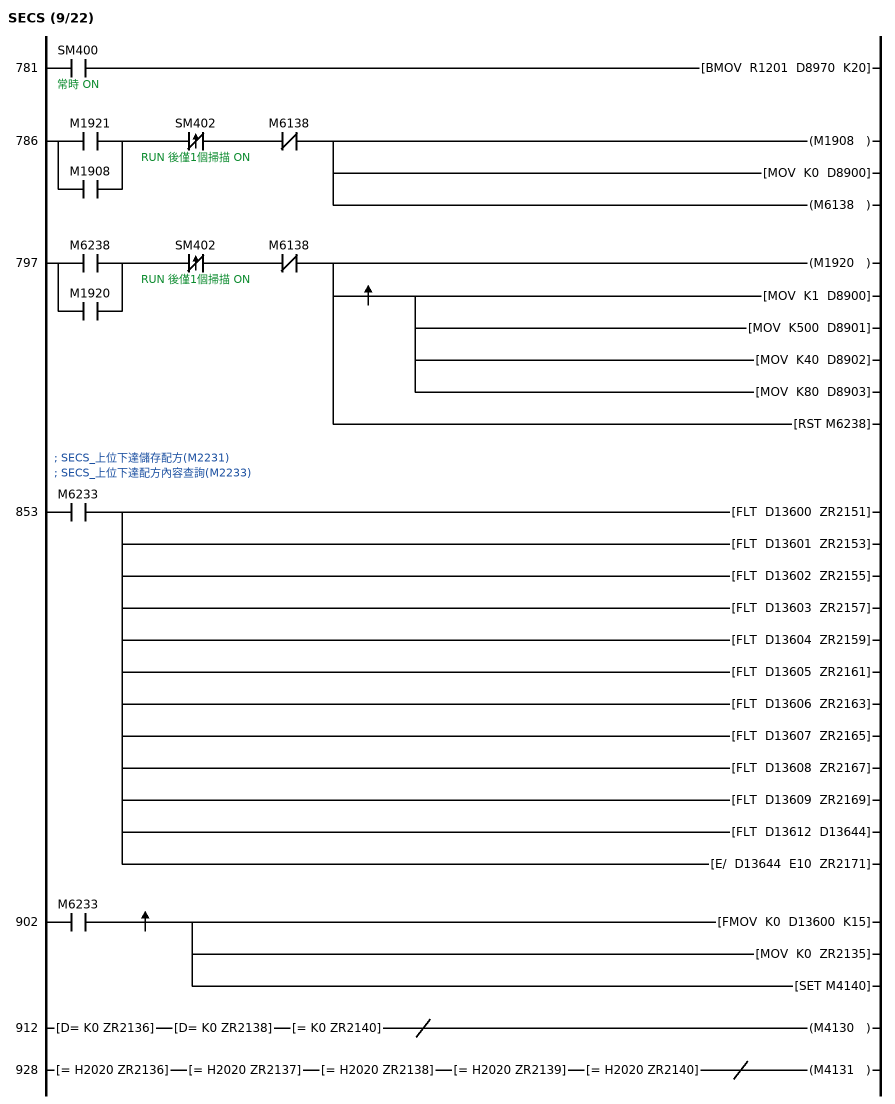
781   LD      SM400  ; 常時 ON
      BMOV    R1201 D8970 K20
786   LD      M1921
      OR      M1908
      ANDPI   SM402  ; RUN 後僅1個掃描 ON
      ANI     M6138
      OUT     M1908
      MOV     K0 D8900
      OUT     M6138
797   LD      M6238
      OR      M1920
      ANDPI   SM402  ; RUN 後僅1個掃描 ON
      ANI     M6138
      OUT     M1920
      MPS
      MEP
      MOV     K1 D8900
      MOV     K500 D8901
      MOV     K40 D8902
      MOV     K80 D8903
      MPP
      RST     M6238
; SECS_上位下達儲存配方(M2231)
; SECS_上位下達配方內容查詢(M2233)
853   LD      M6233
      FLT     D13600 ZR2151
      FLT     D13601 ZR2153
      FLT     D13602 ZR2155
      FLT     D13603 ZR2157
      FLT     D13604 ZR2159
      FLT     D13605 ZR2161
      FLT     D13606 ZR2163
      FLT     D13607 ZR2165
      FLT     D13608 ZR2167
      FLT     D13609 ZR2169
      FLT     D13612 D13644
      E/      D13644 E10 ZR2171
902   LD      M6233
      MEP
      FMOV    K0 D13600 K15
      MOV     K0 ZR2135
      SET     M4140
912   LDD=    K0 ZR2136
      ANDD=   K0 ZR2138
      AND=    K0 ZR2140
      INV
      OUT     M4130
928   LD=     H2020 ZR2136
      AND=    H2020 ZR2137
      AND=    H2020 ZR2138
      AND=    H2020 ZR2139
      AND=    H2020 ZR2140
      INV
      OUT     M4131
